(* IEC 61131-3 sources: lasal-git-demo/CPU/LasalDemoProject/Class/STO081, 1 file *)

(* ---- STO081.st ---- *)
(*!
<Class
	Name               = "STO081"
	Revision           = "1.23"
	RealtimeTask       = "false"
	CyclicTask         = "false"
	BackgroundTask     = "false"
	Sigmatek           = "true"
	OSInterface        = "false"
	HighPriority       = "false"
	Automatic          = "false"
	UpdateMode         = "Prescan"
	IconPath           = ".\Class\sto.ico"
	SharedCommandTable = "true"
	Objectsize         = "(532,120)">
	<Channels>
		<Server Name="Safe_Output1" Visualized="true" Initialize="false" WriteProtected="true" Retentive="false" Comment="State of output (read only)&#13;&#10;&#13;&#10;-1..Error&#13;&#10; 0..Output Low&#13;&#10; 1..Output High"/>
		<Server Name="Safe_Output2" Visualized="true" Initialize="false" WriteProtected="true" Retentive="false" Comment="State of output (read only)&#13;&#10;&#13;&#10;-1..Error&#13;&#10; 0..Output Low&#13;&#10; 1..Output High"/>
		<Server Name="Safe_Output3" Visualized="true" Initialize="false" WriteProtected="true" Retentive="false" Comment="State of output (read only)&#13;&#10;&#13;&#10;-1..Error&#13;&#10; 0..Output Low&#13;&#10; 1..Output High"/>
		<Server Name="Safe_Output4" Visualized="true" Initialize="false" WriteProtected="true" Retentive="false" Comment="State of output (read only)&#13;&#10;&#13;&#10;-1..Error&#13;&#10; 0..Output Low&#13;&#10; 1..Output High"/>
		<Server Name="Safe_Output5" Visualized="true" Initialize="false" WriteProtected="true" Retentive="false" Comment="State of output (read only)&#13;&#10;&#13;&#10;-1..Error&#13;&#10; 0..Output Low&#13;&#10; 1..Output High"/>
		<Server Name="Safe_Output6" Visualized="true" Initialize="false" WriteProtected="true" Retentive="false" Comment="State of output (read only)&#13;&#10;&#13;&#10;-1..Error&#13;&#10; 0..Output Low&#13;&#10; 1..Output High"/>
		<Server Name="Safe_Output7" Visualized="true" Initialize="false" WriteProtected="true" Retentive="false" Comment="State of output (read only)&#13;&#10;&#13;&#10;-1..Error&#13;&#10; 0..Output Low&#13;&#10; 1..Output High"/>
		<Server Name="Safe_Output8" Visualized="true" Initialize="false" WriteProtected="true" Retentive="false" Comment="State of output (read only)&#13;&#10;&#13;&#10;-1..Error&#13;&#10; 0..Output Low&#13;&#10; 1..Output High"/>
		<Server Name="SafeIOError" Visualized="true" Initialize="false" WriteProtected="true" Retentive="false" Comment="Shows which safe outputs are in error.&#13;&#10;The outputs are bitcoded.&#13;&#10;Bit0 = Output1&#13;&#10;Bit1 = Output2&#13;&#10;..."/>
		<Server Name="Unsafe_Output1" Visualized="true" Initialize="true" WriteProtected="false" Retentive="false" Comment="State of output (write only; default value: 0)&#13;&#10;&#13;&#10;If safety is given (output would be 1), you can still switch to zero by writing 0 to this server"/>
		<Server Name="Unsafe_Output2" Visualized="true" Initialize="true" WriteProtected="false" Retentive="false" Comment="State of output (write only; default value: 0)&#13;&#10;&#13;&#10;If safety is given (output would be 1), you can still switch to zero by writing 0 to this server"/>
		<Server Name="Unsafe_Output3" Visualized="true" Initialize="true" WriteProtected="false" Retentive="false" Comment="State of output (write only; default value: 0)&#13;&#10;&#13;&#10;If safety is given (output would be 1), you can still switch to zero by writing 0 to this server"/>
		<Server Name="Unsafe_Output4" Visualized="true" Initialize="true" WriteProtected="false" Retentive="false" Comment="State of output (write only; default value: 0)&#13;&#10;&#13;&#10;If safety is given (output would be 1), you can still switch to zero by writing 0 to this server"/>
		<Server Name="Unsafe_Output5" Visualized="true" Initialize="true" WriteProtected="false" Retentive="false" Comment="State of output (write only; default value: 0)&#13;&#10;&#13;&#10;If safety is given (output would be 1), you can still switch to zero by writing 0 to this server"/>
		<Server Name="Unsafe_Output6" Visualized="true" Initialize="true" WriteProtected="false" Retentive="false" Comment="State of output (write only; default value: 0)&#13;&#10;&#13;&#10;If safety is given (output would be 1), you can still switch to zero by writing 0 to this server"/>
		<Server Name="Unsafe_Output7" Visualized="true" Initialize="true" WriteProtected="false" Retentive="false" Comment="State of output (write only; default value: 0)&#13;&#10;&#13;&#10;If safety is given (output would be 1), you can still switch to zero by writing 0 to this server"/>
		<Server Name="Unsafe_Output8" Visualized="true" Initialize="true" WriteProtected="false" Retentive="false" Comment="State of output (write only; default value: 0)&#13;&#10;&#13;&#10;If safety is given (output would be 1), you can still switch to zero by writing 0 to this server"/>
	</Channels>
	<RevDoku>
		<Owner Company="Sigmatek" Author="SeiChr"/>
		<Dokumentation Revision="1.23" Date="02.06.2021" Author="EisMic" Company="Sigmatek" Description="Added support for analog input modules and showing FW version of safety modules in baseclass."/>
		<Dokumentation Revision="1.22" Date="12.08.2019" Author="LazJos" Company="Sigmatek" Description="Added support for HWAlarms."/>
		<Dokumentation Revision="1.21" Date="08.06.2018" Author="RamAnd" Company="Sigmatek" Description="LASAL Hardware Description (.lhd) file has been updated."/>
		<Dokumentation Revision="1.20" Date="24.04.2018" Author="RamAnd" Company="Sigmatek" Description="Added server to show hardware version if this feature is supported by the safety firmware of the SCP."/>
		<Dokumentation Revision="1.19" Date="30.11.2017" Author="FurDom" Company="Sigmatek" Description="Added QuitComError server description to .lhd file"/>
		<Dokumentation Revision="1.18" Date="24.10.2016" Author="ZoePat" Company="Sigmatek" Description="Set the base class to visualized, so the embedded string object &quot;SerialNoStr&quot; can be used in the LSE."/>
		<Dokumentation Revision="1.17" Date="12.07.2016" Author="SeiChr" Company="Sigmatek" Description="Added Values for the total Current calculation. SA 31571"/>
		<Dokumentation Revision="1.16" Date="21.01.2016" Author="EisMic" Company="Sigmatek" Description="Outputs are now written in RtPostScan instead of RtPreScan to improve the reaction speed."/>
		<Dokumentation Revision="1.15" Date="16.04.2015" Author="EisMic" Company="Sigmatek" Description="Added support for graphical hardware editor."/>
		<Dokumentation Revision="1.14" Date="31.10.2014" Author="lanste" Company="Sigmatek" Description="Fixed error: Safe IO were displayed on wrong safety hardwareclass if the class is not required and not online.&#13;&#10;Fixed error: Safe IO were displayed on wrong safety hardwareclass if the hardware configuration did not match the project configuration.&#13;&#10;Set IOs to -2 if Class is not online."/>
		<Dokumentation Revision="1.13" Date="31.07.2014" Author="PieSte" Company="Sigmatek" Description="Added QuitComError server to quit errors on safety cpu."/>
		<Dokumentation Revision="1.12" Date="24.04.2014" Author="RamAnd" Company="Sigmatek" Description="Clear module info at the servers if a disconnect event occurs."/>
		<Dokumentation Revision="1.11" Date="28.03.2014" Author="EisMic" Company="Sigmatek" Description="Added server RetryCounteruC1 and RetryCounteruC2."/>
		<Dokumentation Revision="1.10" Date="22.01.2014" Author="RamAnd&#13;&#10;LanSte" Company="Sigmatek" Description="Added functionality to use module optional via define DEACTIVATED_LSL as Place value.&#13;&#10;Read Client Required and Place in Init SdiasSafetyBase"/>
		<Dokumentation Revision="1.0" Date="04.12.2013" Author="RamAnd" Company="Sigmatek" Description="First library version"/>
	</RevDoku>
	<Network Name="STO081">
		<!-- List of Components in this network -->
		<Components>
			<Object
				Name       = "_base"
				Class      = "SdiasSafetyBase"
				Position   = "(218,120)"
				Visualized = "true">
				<Channels>
					<Server Name="CallCommand"/>
					<Server Name="ClassState"/>
					<Server Name="DeviceID"/>
					<Server Name="FWVersion"/>
					<Server Name="HwVersion"/>
					<Server Name="QuitComError"/>
					<Server Name="RetryCounteruC1"/>
					<Server Name="RetryCounteruC2"/>
					<Server Name="SafetyNumber"/>
					<Server Name="SerialNo"/>
					<Client Name="AnalogInputBytesNeeded"/>
					<Client Name="InputsNeeded" Value="0"/>
					<Client Name="OutputsNeeded" Value="8"/>
					<Client Name="Place"/>
					<Client Name="Required" Value="1"/>
					<Client Name="SdiasSafetyIn"/>
					<Client Name="SetDeviceID" Value="2#00010001"/>
					<Client Name="toStdLib"/>
				</Channels>
			</Object>
		</Components>
		<Comments>
		</Comments>
		<!-- List of Connections in this network -->
		<Connections>
			<Connection Source="this.ClassState" Destination="_base.ClassState" Vertices="(992,210),(820,210),"/>
			<Connection Source="_base.SdiasSafetyIn" Destination="this.SdiasSafetyIn" Vertices="(218,210),(38,210),"/>
			<Connection Source="_base.Place" Destination="this.Place" Vertices="(218,270),(38,270),"/>
			<Connection Source="this.DeviceID" Destination="_base.DeviceID" Vertices="(992,270),(820,270),"/>
			<Connection Source="_base.Required" Destination="this.Required" Vertices="(218,330),(38,330),"/>
			<Connection Source="this.SerialNo" Destination="_base.SerialNo" Vertices="(992,390),(820,450),"/>
			<Connection Source="this.SafetyNumber" Destination="_base.SafetyNumber" Vertices="(992,450),(820,510),"/>
			<Connection Source="this.RetryCounteruC1" Destination="_base.RetryCounteruC1" Vertices="(992,510),(820,570),"/>
			<Connection Source="this.RetryCounteruC2" Destination="_base.RetryCounteruC2" Vertices="(992,570),(820,630),"/>
			<Connection Source="this.QuitComError" Destination="_base.QuitComError" Vertices="(992,630),(820,750),"/>
			<Connection Source="this.HwVersion" Destination="_base.HwVersion" Vertices="(992,330),(820,330),"/>
		</Connections>
		<!-- Headerfiles -->
		<Options>
		</Options>
	</Network>
</Class>
*)
#pragma using SdiasSafetyBase

STO081 : CLASS
: SdiasSafetyBase
  //Servers:
	Safe_Output1 	: SvrCh_DINT;
	Unsafe_Output1 	: SvrCh_DINT;
	Safe_Output2 	: SvrCh_DINT;
	Unsafe_Output2 	: SvrCh_DINT;
	Safe_Output3 	: SvrCh_DINT;
	Unsafe_Output3 	: SvrCh_DINT;
	Safe_Output4 	: SvrCh_DINT;
	Unsafe_Output4 	: SvrCh_DINT;
	Safe_Output5 	: SvrCh_DINT;
	Unsafe_Output5 	: SvrCh_DINT;
	Safe_Output6 	: SvrCh_DINT;
	Unsafe_Output6 	: SvrCh_DINT;
	Safe_Output7 	: SvrCh_DINT;
	Unsafe_Output7 	: SvrCh_DINT;
	Safe_Output8 	: SvrCh_DINT;
	Unsafe_Output8 	: SvrCh_DINT;
	SafeIOError 	: SvrCh_BDINT;
  //Clients:
  //Variables:
  //Functions:

	FUNCTION VIRTUAL GLOBAL Init;

	FUNCTION VIRTUAL GLOBAL RtWork
		VAR_INPUT
			EAX 	: UDINT;
		END_VAR
		VAR_OUTPUT
			state (EAX) 	: UDINT;
		END_VAR;
				//! <Function Comment="Called when class state was set to _NoHardware &#13;&#10;No Implementation Overload in derived classes if needed " Name="SetClassStateError"/>
	FUNCTION VIRTUAL SetClassStateError;

	FUNCTION VIRTUAL GLOBAL Unsafe_Output1::Write
		VAR_INPUT
			input (EAX) 	: DINT;
		END_VAR
		VAR_OUTPUT
			result (EAX) 	: DINT;
		END_VAR;

	FUNCTION VIRTUAL GLOBAL Unsafe_Output2::Write
		VAR_INPUT
			input (EAX) 	: DINT;
		END_VAR
		VAR_OUTPUT
			result (EAX) 	: DINT;
		END_VAR;

	FUNCTION VIRTUAL GLOBAL Unsafe_Output3::Write
		VAR_INPUT
			input (EAX) 	: DINT;
		END_VAR
		VAR_OUTPUT
			result (EAX) 	: DINT;
		END_VAR;

	FUNCTION VIRTUAL GLOBAL Unsafe_Output4::Write
		VAR_INPUT
			input (EAX) 	: DINT;
		END_VAR
		VAR_OUTPUT
			result (EAX) 	: DINT;
		END_VAR;

	FUNCTION VIRTUAL GLOBAL Unsafe_Output5::Write
		VAR_INPUT
			input (EAX) 	: DINT;
		END_VAR
		VAR_OUTPUT
			result (EAX) 	: DINT;
		END_VAR;

	FUNCTION VIRTUAL GLOBAL Unsafe_Output6::Write
		VAR_INPUT
			input (EAX) 	: DINT;
		END_VAR
		VAR_OUTPUT
			result (EAX) 	: DINT;
		END_VAR;

	FUNCTION VIRTUAL GLOBAL Unsafe_Output7::Write
		VAR_INPUT
			input (EAX) 	: DINT;
		END_VAR
		VAR_OUTPUT
			result (EAX) 	: DINT;
		END_VAR;

	FUNCTION VIRTUAL GLOBAL Unsafe_Output8::Write
		VAR_INPUT
			input (EAX) 	: DINT;
		END_VAR
		VAR_OUTPUT
			result (EAX) 	: DINT;
		END_VAR;
  //Tables:
	FUNCTION @STD
		VAR_OUTPUT
			ret_code	: CONFSTATES;
		END_VAR;
	FUNCTION GLOBAL TAB @CT_;
END_CLASS;

FUNCTION VIRTUAL GLOBAL STO081::RtWork
	VAR_INPUT
		EAX 	: UDINT;
	END_VAR
	VAR_OUTPUT
		state (EAX) 	: UDINT;
	END_VAR

  // 0 = inputs, 1 = outputs
  if EAX then

    // if AcceptState bit is set => accept state
    if IOStates AND 2#10 then
      Safe_Output1 := to_dint(IOStates AND 2#1);

      // show error state of this IO
      SafeIOError.1 := FALSE;
    else
      // otherwise, there's an error
      Safe_Output1 := -1;

      // show error state of this IO
      SafeIOError.1 := TRUE;
    end_if;

    // if AcceptState bit is set => accept state
    if IOStates AND 2#1000 then
      Safe_Output2 := to_dint(IOStates AND 2#100) SHR 2;

      // show error state of this IO
      SafeIOError.2 := FALSE;
    else
      // otherwise, there's an error
      Safe_Output2 := -1;

      // show error state of this IO
      SafeIOError.2 := TRUE;
    end_if;

    // if AcceptState bit is set => accept state
    if IOStates AND 2#100000 then
      Safe_Output3 := to_dint(IOStates AND 2#10000) SHR 4;

      // show error state of this IO
      SafeIOError.3 := FALSE;
    else
      // otherwise, there's an error
      Safe_Output3 := -1;

      // show error state of this IO
      SafeIOError.3 := TRUE;
    end_if;

    // if AcceptState bit is set => accept state
    if IOStates AND 2#10000000 then
      Safe_Output4 := to_dint(IOStates AND 2#1000000) SHR 6;

      // show error state of this IO
      SafeIOError.4 := FALSE;
    else
      // otherwise, there's an error
      Safe_Output4 := -1;

      // show error state of this IO
      SafeIOError.4 := TRUE;
    end_if;

    // if AcceptState bit is set => accept state
    if IOStates AND 2#1000000000 then
      Safe_Output5 := to_dint(IOStates AND 2#100000000) SHR 8;

      // show error state of this IO
      SafeIOError.5 := FALSE;
    else
      // otherwise, there's an error
      Safe_Output5 := -1;

      // show error state of this IO
      SafeIOError.5 := TRUE;
    end_if;

    // if AcceptState bit is set => accept state
    if IOStates AND 2#100000000000 then
      Safe_Output6 := to_dint(IOStates AND 2#10000000000) SHR 10;

      // show error state of this IO
      SafeIOError.6 := FALSE;
    else
      // otherwise, there's an error
      Safe_Output6 := -1;

      // show error state of this IO
      SafeIOError.6 := TRUE;
    end_if;

    // if AcceptState bit is set => accept state
    if IOStates AND 2#10000000000000 then
      Safe_Output7 := to_dint(IOStates AND 2#1000000000000) SHR 12;

      // show error state of this IO
      SafeIOError.7 := FALSE;
    else
      // otherwise, there's an error
      Safe_Output7 := -1;

      // show error state of this IO
      SafeIOError.7 := TRUE;
    end_if;

    // if AcceptState bit is set => accept state
    if IOStates AND 2#1000000000000000 then
      Safe_Output8 := to_dint(IOStates AND 2#100000000000000) SHR 14;

      // show error state of this IO
      SafeIOError.8 := FALSE;
    else
      // otherwise, there's an error
      Safe_Output8 := -1;

      // show error state of this IO
      SafeIOError.8 := TRUE;
    end_if;
  end_if;

	state := READY;

END_FUNCTION

FUNCTION VIRTUAL GLOBAL STO081::Unsafe_Output1::Write
	VAR_INPUT
		input (EAX) 	: DINT;
	END_VAR
	VAR_OUTPUT
		result (EAX) 	: DINT;
	END_VAR

  if input then
    result := Unsafe_Output1 := 1;
    UnsafeOutputStates.1 := TRUE;
  else
    result := Unsafe_Output1 := 0;
    UnsafeOutputStates.1 := FALSE;
  end_if;

END_FUNCTION

FUNCTION VIRTUAL GLOBAL STO081::Unsafe_Output2::Write
	VAR_INPUT
		input (EAX) 	: DINT;
	END_VAR
	VAR_OUTPUT
		result (EAX) 	: DINT;
	END_VAR

  if input then
    result := Unsafe_Output2 := 1;
    UnsafeOutputStates.2 := TRUE;
  else
    result := Unsafe_Output2 := 0;
    UnsafeOutputStates.2 := FALSE;
  end_if;

END_FUNCTION

FUNCTION VIRTUAL GLOBAL STO081::Unsafe_Output3::Write
	VAR_INPUT
		input (EAX) 	: DINT;
	END_VAR
	VAR_OUTPUT
		result (EAX) 	: DINT;
	END_VAR

  if input then
    result := Unsafe_Output3 := 1;
    UnsafeOutputStates.3 := TRUE;
  else
    result := Unsafe_Output3 := 0;
    UnsafeOutputStates.3 := FALSE;
  end_if;

END_FUNCTION

FUNCTION VIRTUAL GLOBAL STO081::Unsafe_Output4::Write
	VAR_INPUT
		input (EAX) 	: DINT;
	END_VAR
	VAR_OUTPUT
		result (EAX) 	: DINT;
	END_VAR

  if input then
    result := Unsafe_Output4 := 1;
    UnsafeOutputStates.4 := TRUE;
  else
    result := Unsafe_Output4 := 0;
    UnsafeOutputStates.4 := FALSE;
  end_if;

END_FUNCTION

FUNCTION VIRTUAL GLOBAL STO081::Unsafe_Output5::Write
	VAR_INPUT
		input (EAX) 	: DINT;
	END_VAR
	VAR_OUTPUT
		result (EAX) 	: DINT;
	END_VAR

  if input then
    result := Unsafe_Output5 := 1;
    UnsafeOutputStates.5 := TRUE;
  else
    result := Unsafe_Output5 := 0;
    UnsafeOutputStates.5 := FALSE;
  end_if;

END_FUNCTION

FUNCTION VIRTUAL GLOBAL STO081::Unsafe_Output6::Write
	VAR_INPUT
		input (EAX) 	: DINT;
	END_VAR
	VAR_OUTPUT
		result (EAX) 	: DINT;
	END_VAR

  if input then
    result := Unsafe_Output6 := 1;
    UnsafeOutputStates.6 := TRUE;
  else
    result := Unsafe_Output6 := 0;
    UnsafeOutputStates.6 := FALSE;
  end_if;

END_FUNCTION

FUNCTION VIRTUAL GLOBAL STO081::Unsafe_Output7::Write
	VAR_INPUT
		input (EAX) 	: DINT;
	END_VAR
	VAR_OUTPUT
		result (EAX) 	: DINT;
	END_VAR

  if input then
    result := Unsafe_Output7 := 1;
    UnsafeOutputStates.7 := TRUE;
  else
    result := Unsafe_Output7 := 0;
    UnsafeOutputStates.7 := FALSE;
  end_if;

END_FUNCTION

FUNCTION VIRTUAL GLOBAL STO081::Unsafe_Output8::Write
	VAR_INPUT
		input (EAX) 	: DINT;
	END_VAR
	VAR_OUTPUT
		result (EAX) 	: DINT;
	END_VAR

  if input then
    result := Unsafe_Output8 := 1;
    UnsafeOutputStates.8 := TRUE;
  else
    result := Unsafe_Output8 := 0;
    UnsafeOutputStates.8 := FALSE;
  end_if;

END_FUNCTION

FUNCTION VIRTUAL GLOBAL STO081::Init

  SdiasSafetyBase::Init();

  if us_FirstScan = 1 then
    Unsafe_Output1 := Unsafe_Output1 <> 0;
    Unsafe_Output2 := Unsafe_Output2 <> 0;
    Unsafe_Output3 := Unsafe_Output3 <> 0;
    Unsafe_Output4 := Unsafe_Output4 <> 0;
    Unsafe_Output5 := Unsafe_Output5 <> 0;
    Unsafe_Output6 := Unsafe_Output6 <> 0;
    Unsafe_Output7 := Unsafe_Output7 <> 0;
    Unsafe_Output8 := Unsafe_Output8 <> 0;

    UnsafeOutputStates.1 := to_bool(Unsafe_Output1);
    UnsafeOutputStates.2 := to_bool(Unsafe_Output2);
    UnsafeOutputStates.3 := to_bool(Unsafe_Output3);
    UnsafeOutputStates.4 := to_bool(Unsafe_Output4);
    UnsafeOutputStates.5 := to_bool(Unsafe_Output5);
    UnsafeOutputStates.6 := to_bool(Unsafe_Output6);
    UnsafeOutputStates.7 := to_bool(Unsafe_Output7);
    UnsafeOutputStates.8 := to_bool(Unsafe_Output8);
  end_if;

END_FUNCTION

FUNCTION VIRTUAL STO081::SetClassStateError
  VAR
    i : UDINT;
    pServer : ^DINT;
  END_VAR

  pServer := #Safe_Output1;

  for i := 0 to 7 do
    pServer^ := SDIAS_SAFETY_INVALID_IO_NOHW;
    pServer += sizeof(SvrCh) * 2;
  end_for;
END_FUNCTION
